FUNCTION_BLOCK Utilidades_1
VAR_INPUT
END_VAR
VAR_OUTPUT
END_VAR
VAR
	
END_VAR

GVL_Funciones_Paro.Temporizador1min(IN:=not GVL_Funciones_Paro.Temporizador1min.Q , PT:= T#60s, Q=> , ET=> );

END_FUNCTION_BLOCK

(* stored: Version 1.1.0.1, ProductVersion 3.1.4024.12
   POU Utilidades_1: Id {6888e73a-9c15-48f8-a680-93406fd4e4af}, SpecialFunc None *)
